(* CoDeSys 2.3.9.19 project: md_roman.pro *)
(* Libraries: D:\_wago\library\PowerMeasurement_01.lib 28.1.08 13:32:32, SysLibTime.lib 5.10.04 10:39:34, D:\_wago\library\Dali_01eng.lib 6.2.07 12:38:12, Building_common.lib 15.5.09 13:11:15, Util.lib 1.6.07 09:40:58, Standard.lib 22.11.04 11:21:12, SYSLIBCALLBACK.LIB 20.4.05 11:04:48 *)

(* PLC configuration (modules and I/O channels)
TL01 AT %IX17.0 [BOOLOnX_I] Vypinac_sklad_sklad
TL02 AT %IX17.1 [BOOLOnX_I] Vypinac_sklad_prodejna
TL03 AT %IX17.2 [BOOLOnX_I] Vypinac_sklad_z_venku
TL04 AT %IX17.3 [BOOLOnX_I] Vypinac_sklad_vrata_predni
TL05 AT %IX17.4 [BOOLOnX_I] Vypinac_sklad_vrata_zadni
TL06 AT %IX17.5 [BOOLOnX_I] Vypinac_prodejna_kolotoc_sude
TL07 AT %IX17.6 [BOOLOnX_I] Vypinac_prodejna_kolotoc_liche
TL08 AT %IX17.7 [BOOLOnX_I] Vypinac_prodejna_vypinac
TL09 AT %IX17.8 [BOOLOnX_I] Prodejna_Dali
TL10 AT %IX17.9 [BOOLOnX_I] Prodejna_faugule_OUT13
TL11 AT %IX17.10 [BOOLOnX_I] Ch_3 Digital input
TL12 AT %IX17.11 [BOOLOnX_I] Ch_4 Digital input
TL13 AT %IX17.12 [BOOLOnX_I] Ch_5 Digital input
AT %IX17.13 [BOOLOnX_I] Ch_6 Digital input
AT %IX17.14 [BOOLOnX_I] Ch_7 Digital input
AT %IX17.15 [BOOLOnX_I] Ch_8 Digital input
0750-0430 8 DI 24 V DC 3.0ms [Type_1_8_Channels] node 2, in %IB2 out %QB2 {INTTypePAAssignment = PLC; INTTypeModule = plugged}
  AT %IX18.0 [BOOLOnX_I] Ch_1 Digital input
  AT %IX18.1 [BOOLOnX_I] Ch_2 Digital input
  AT %IX18.2 [BOOLOnX_I] Ch_3 Digital input
  AT %IX18.3 [BOOLOnX_I] Ch_4 Digital input
  AT %IX18.4 [BOOLOnX_I] Ch_5 Digital input
  AT %IX18.5 [BOOLOnX_I] Ch_6 Digital input
  AT %IX18.6 [BOOLOnX_I] Ch_7 Digital input
  AT %IX18.7 [BOOLOnX_I] Ch_8 Digital input
0750-0530 8 DO 24 V DC 0.5A [Type_10_8_Channels] node 3, in %IB3 out %QB3 {INTTypePAAssignment = PLC; INTTypeModule = plugged}
  KA01 AT %QX9.0 [BOOLOnX_Q] Nevim
  KA02 AT %QX9.1 [BOOLOnX_Q] kolotoc2
  KA03 AT %QX9.2 [BOOLOnX_Q] kolotoc3
  KA04 AT %QX9.3 [BOOLOnX_Q] kolotoc4
  KA05 AT %QX9.4 [BOOLOnX_Q] kolotoc5
  KA06 AT %QX9.5 [BOOLOnX_Q] kolotoc6
  KA07 AT %QX9.6 [BOOLOnX_Q] kolotoc7
  KA08 AT %QX9.7 [BOOLOnX_Q] kolotoc8
0750-0530 8 DO 24 V DC 0.5A [Type_10_8_Channels] node 4, in %IB4 out %QB4 {INTTypePAAssignment = PLC; INTTypeModule = plugged}
  KA09 AT %QX9.8 [BOOLOnX_Q] kolotoc9
  KA10 AT %QX9.9 [BOOLOnX_Q] kolotoc10
  KA11 AT %QX9.10 [BOOLOnX_Q] kolotoc11
  KA12 AT %QX9.11 [BOOLOnX_Q] kolotoc12
  KA13 AT %QX9.12 [BOOLOnX_Q] svetlo_vchod_do_prodejny
  KA14 AT %QX9.13 [BOOLOnX_Q] reklama
  KA15 AT %QX9.14 [BOOLOnX_Q] svetlo_vrata_predni
  KA16 AT %QX9.15 [BOOLOnX_Q] svetlo_vrata_zadni
0750-0530 8 DO 24 V DC 0.5A [Type_10_8_Channels] node 5, in %IB5 out %QB5 {INTTypePAAssignment = PLC; INTTypeModule = plugged}
  KA17 AT %QX10.0 [BOOLOnX_Q] Ch_1 Digital output
  AT %QX10.1 [BOOLOnX_Q] Ch_2 Digital output
  AT %QX10.2 [BOOLOnX_Q] Ch_3 Digital output
  KA20 AT %QX10.3 [BOOLOnX_Q] Ch_4 Digital output
  AT %QX10.4 [BOOLOnX_Q] Ch_5 Digital output
  AT %QX10.5 [BOOLOnX_Q] Ch_6 Digital output
  AT %QX10.6 [BOOLOnX_Q] Ch_7 Digital output
  AT %QX10.7 [BOOLOnX_Q] Ch_8 Digital output
0750-0530 8 DO 24 V DC 0.5A [Type_10_8_Channels] node 6, in %IB6 out %QB6 {INTTypePAAssignment = PLC; INTTypeModule = plugged}
  AT %QX10.8 [BOOLOnX_Q] Ch_1 Digital output
  AT %QX10.9 [BOOLOnX_Q] Ch_2 Digital output
  AT %QX10.10 [BOOLOnX_Q] Ch_3 Digital output
  AT %QX10.11 [BOOLOnX_Q] Ch_4 Digital output
  AT %QX10.12 [BOOLOnX_Q] Ch_5 Digital output
  AT %QX10.13 [BOOLOnX_Q] Ch_6 Digital output
  AT %QX10.14 [BOOLOnX_Q] Ch_7 Digital output
  AT %QX10.15 [BOOLOnX_Q] Ch_8 Digital output
Analog_1 AT %IW0 [WORDOnW_I] Ch_1 Input word
AT %IW1 [WORDOnW_I] Ch_2 Input word
AT %IW2 [WORDOnW_I] Ch_3 Input word
AT %IW3 [WORDOnW_I] Ch_4 Input word
Teplota_1 AT %IW4 [INTOnW_I] Ch_1 signed Input value
Teplota_2 AT %IW5 [INTOnW_I] Ch_2 signed Input value
Teplota_3 AT %IW6 [INTOnW_I] Ch_3 signed Input value
Teplota_4 AT %IW7 [INTOnW_I] Ch_4 signed Input value
0750-0641 DALI/DSI-Master [Type_36_1_Channels] node 9, in %IB9 out %QB9 {INTTypePAAssignment = PLC; INTTypeModule = plugged}
  AT %IX8.0 [BOOLOnX_I] Transmit accepted
  AT %IX8.1 [BOOLOnX_I] Receive request
  AT %IX8.2 [BOOLOnX_I] Init accepted
  AT %IX8.3 [BOOLOnX_I] Actor Error
  AT %IX8.4 [BOOLOnX_I] Frame Error
  AT %IX8.5 [BOOLOnX_I] Bus Error
  AT %IX8.6 [BOOLOnX_I] General Module Error
  AT %IB17 [BYTEOnB_I] DALI Response
  AT %IB18 [BYTEOnB_I] DALI Address
  AT %IB19 [BYTEOnB_I] Message 3
  AT %IB20 [BYTEOnB_I] Message 2
  AT %IB21 [BYTEOnB_I] Message 1
  AT %QX0.0 [BOOLOnX_Q] Transmit request
  AT %QX0.1 [BOOLOnX_Q] Receive accepted
  AT %QX0.2 [BOOLOnX_Q] Init request
  AT %QB1 [BYTEOnB_Q] DALI Command, DSI dimming value
  AT %QB2 [BYTEOnB_Q] DALI Address
  AT %QB3 [BYTEOnB_Q] Parameter 2
  AT %QB4 [BYTEOnB_Q] Parameter 1
  AT %QB5 [BYTEOnB_Q] Command extension
fazeVstup AT %IB22 [BYTEOnB_I] First Byte of 12
fazeVystup AT %QB6 [BYTEOnB_Q] First Byte of 12
Fieldbus variables [FB_VARS] node 1, in %IB0 out %QB0
*)

(* Task configuration *)
TASK hlavni (PRIORITY := 1, INTERVAL := T#20ms);
	PLC_PRG();
END_TASK

(* Global variable list: Global_Variables *)
VAR_GLOBAL
	start_bit: BOOL;
	Inicialiazace_DALI: BOOL;
	Inicializuj: BOOL;
	TL08s: BOOL;
	TL07s: BOOL;
	TL10s: BOOL;
	TL06s: BOOL;
	TL05s: BOOL;
	TL01s: BOOL;
	TL09s: BOOL;
END_VAR

(* POU PLC_PRG, FBD *)
PROGRAM PLC_PRG
VAR
	cas_datum: CurTimeEx;
	System_cas: SysTime64;
	System_datum: SystemTimeDate;
	kolotoc1: kolotoc;
	kolotoc2: kolotoc;
	BLINK_nouzaky: BLINK;
	LibovolnyVystup: BOOL;
END_VAR
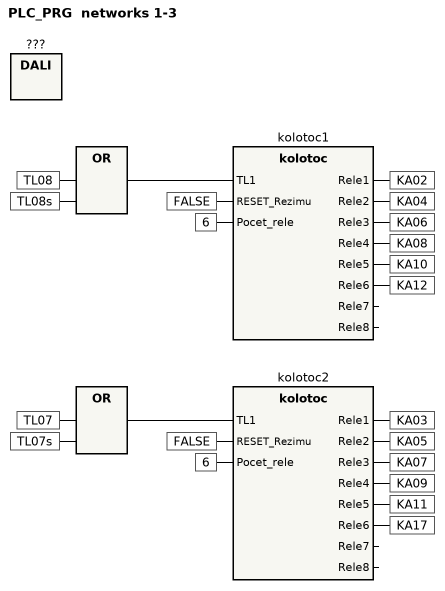
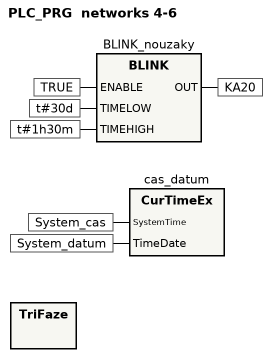
_FBD_ (* Function Block Diagram *)
NETWORK 1
	???:DALI()
NETWORK 2
	kolotoc1:kolotoc(TL1: OR(TL08, TL08s), RESET_Rezimu: FALSE, Pocet_rele: 6, Rele2 => KA04, Rele3 => KA06, Rele4 => KA08, Rele5 => KA10, Rele6 => KA12) => KA02
NETWORK 3
	kolotoc2:kolotoc(TL1: OR(TL07, TL07s), RESET_Rezimu: FALSE, Pocet_rele: 6, Rele2 => KA05, Rele3 => KA07, Rele4 => KA09, Rele5 => KA11, Rele6 => KA17) => KA03
NETWORK 4
	BLINK_nouzaky:BLINK(ENABLE: TRUE, TIMELOW: t#30d, TIMEHIGH: t#1h30m) => KA20
NETWORK 5
	cas_datum:CurTimeEx(SystemTime: System_cas, TimeDate: System_datum)
NETWORK 6
	TriFaze()
_END_FBD_
(* the same logic as Structured Text *)
(* Network 1: see the listing above *)
(* Network 2 *)
kolotoc1(TL1 := TL08 OR TL08s, RESET_Rezimu := FALSE, Pocet_rele := 6);
KA04 := kolotoc1.Rele2;
KA06 := kolotoc1.Rele3;
KA08 := kolotoc1.Rele4;
KA10 := kolotoc1.Rele5;
KA12 := kolotoc1.Rele6;
KA02 := kolotoc1.Rele1;
(* Network 3 *)
kolotoc2(TL1 := TL07 OR TL07s, RESET_Rezimu := FALSE, Pocet_rele := 6);
KA05 := kolotoc2.Rele2;
KA07 := kolotoc2.Rele3;
KA09 := kolotoc2.Rele4;
KA11 := kolotoc2.Rele5;
KA17 := kolotoc2.Rele6;
KA03 := kolotoc2.Rele1;
(* Network 4 *)
BLINK_nouzaky(ENABLE := TRUE, TIMELOW := t#30d, TIMEHIGH := t#1h30m);
KA20 := BLINK_nouzaky.OUT;
(* Network 5 *)
cas_datum(SystemTime := System_cas, TimeDate := System_datum);
(* Network 6 *)
TriFaze();
END_PROGRAM

(* POU dali/kolotoc, FBD *)
FUNCTION_BLOCK kolotoc
VAR
	Data_platna: BOOL;
	Data_platna_reset: BOOL;
	T_Data_platna: TON;
	T_Data_platna_reset: TON;
	Stisk_kratky: BOOL := FALSE;
	Stisk_dlouhy: BOOL := FALSE;
	T_stisk_TLx: TON;
	F_trig_hr1: F_TRIG;
	R_trig_hr2: R_TRIG;
	TL1_Citac: CTU;
	SR_stisk_TLx: SR;
	ZAP_VYP: BOOL;




	TP_byl_kratky: TP;
	Q_byl_kratky: BOOL;
	blok_kratky: BOOL;
	TL1_hr1: BOOL;
	SET_stisk_TL1: BOOL;
	Q_stisk_TL1: BOOL;
	TL1_INT: INT;
END_VAR

VAR_OUTPUT
	Rele1: BOOL;
	Rele2: BOOL;
	Rele3: BOOL;
	Rele4: BOOL;
	Rele5: BOOL;
	Rele6: BOOL;
	Rele7: BOOL;
	Rele8: BOOL;
END_VAR
VAR_INPUT
	TL1: BOOL;
	RESET_Rezimu: BOOL;
	Pocet_rele: INT;
END_VAR
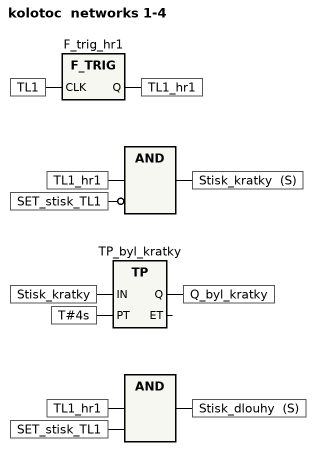
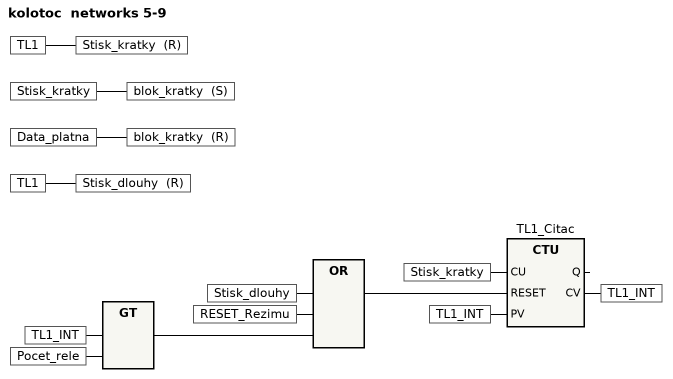
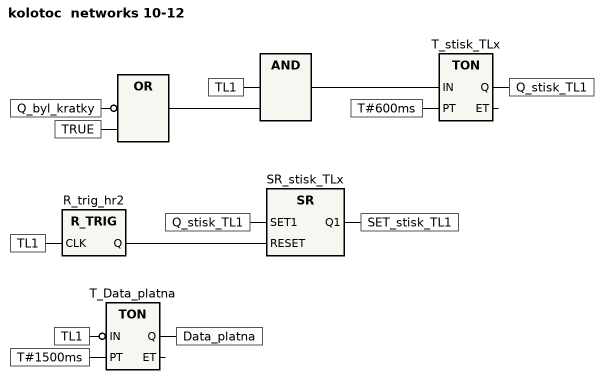
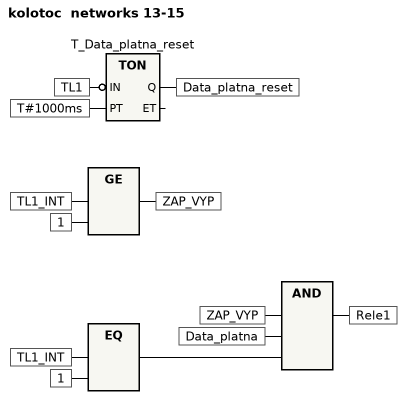
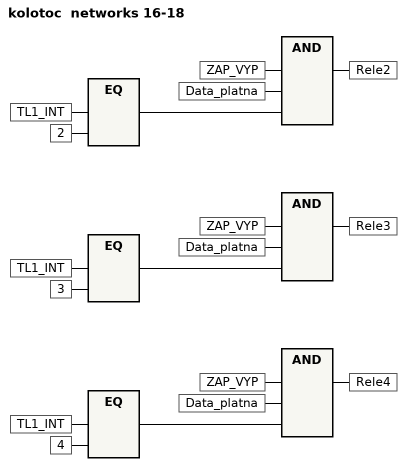
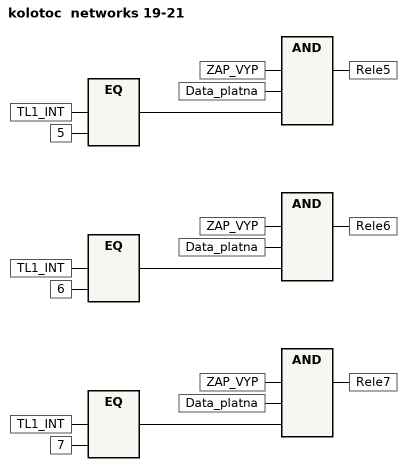
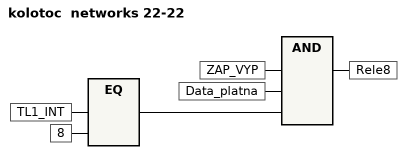
_FBD_ (* Function Block Diagram *)
NETWORK 1
	F_trig_hr1:F_TRIG(CLK: TL1) => TL1_hr1
NETWORK 2
	AND(TL1_hr1, NOT SET_stisk_TL1) => S Stisk_kratky
NETWORK 3
	TP_byl_kratky:TP(IN: Stisk_kratky, PT: T#4s) => Q_byl_kratky
NETWORK 4
	AND(TL1_hr1, SET_stisk_TL1) => S Stisk_dlouhy
NETWORK 5
	TL1 => R Stisk_kratky
NETWORK 6
	Stisk_kratky => S blok_kratky
NETWORK 7
	Data_platna => R blok_kratky
NETWORK 8
	TL1 => R Stisk_dlouhy
NETWORK 9
	TL1_Citac:CTU(CU: Stisk_kratky, RESET: OR(Stisk_dlouhy, RESET_Rezimu, GT(TL1_INT, Pocet_rele)), PV: TL1_INT, CV => TL1_INT)
NETWORK 10 (* delka stisku TLx *)
	T_stisk_TLx:TON(IN: AND(TL1, OR(NOT Q_byl_kratky, TRUE)), PT: T#600ms) => Q_stisk_TL1
NETWORK 11
	SR_stisk_TLx:SR(SET1: Q_stisk_TL1, RESET: R_trig_hr2:R_TRIG(CLK: TL1)) => SET_stisk_TL1
NETWORK 12 (* Data platna *)
	T_Data_platna:TON(IN: NOT TL1, PT: T#1500ms) => Data_platna
NETWORK 13 (* Data platna *)
	T_Data_platna_reset:TON(IN: NOT TL1, PT: T#1000ms) => Data_platna_reset
NETWORK 14
	GE(TL1_INT, 1) => ZAP_VYP
NETWORK 15
	AND(ZAP_VYP, Data_platna, EQ(TL1_INT, 1)) => Rele1
NETWORK 16
	AND(ZAP_VYP, Data_platna, EQ(TL1_INT, 2)) => Rele2
NETWORK 17
	AND(ZAP_VYP, Data_platna, EQ(TL1_INT, 3)) => Rele3
NETWORK 18
	AND(ZAP_VYP, Data_platna, EQ(TL1_INT, 4)) => Rele4
NETWORK 19
	AND(ZAP_VYP, Data_platna, EQ(TL1_INT, 5)) => Rele5
NETWORK 20
	AND(ZAP_VYP, Data_platna, EQ(TL1_INT, 6)) => Rele6
NETWORK 21
	AND(ZAP_VYP, Data_platna, EQ(TL1_INT, 7)) => Rele7
NETWORK 22
	AND(ZAP_VYP, Data_platna, EQ(TL1_INT, 8)) => Rele8
_END_FBD_
(* the same logic as Structured Text *)
(* Network 1 *)
F_trig_hr1(CLK := TL1);
TL1_hr1 := F_trig_hr1.Q;
(* Network 2 *)
IF TL1_hr1 AND NOT SET_stisk_TL1 THEN Stisk_kratky := TRUE; END_IF;
(* Network 3 *)
TP_byl_kratky(IN := Stisk_kratky, PT := T#4s);
Q_byl_kratky := TP_byl_kratky.Q;
(* Network 4 *)
IF TL1_hr1 AND SET_stisk_TL1 THEN Stisk_dlouhy := TRUE; END_IF;
(* Network 5 *)
IF TL1 THEN Stisk_kratky := FALSE; END_IF;
(* Network 6 *)
IF Stisk_kratky THEN blok_kratky := TRUE; END_IF;
(* Network 7 *)
IF Data_platna THEN blok_kratky := FALSE; END_IF;
(* Network 8 *)
IF TL1 THEN Stisk_dlouhy := FALSE; END_IF;
(* Network 9 *)
TL1_Citac(CU := Stisk_kratky, RESET := Stisk_dlouhy OR RESET_Rezimu OR (TL1_INT > Pocet_rele), PV := TL1_INT);
TL1_INT := TL1_Citac.CV;
(* Network 10: see the listing above *)
(* Network 11 *)
R_trig_hr2(CLK := TL1);
SR_stisk_TLx(SET1 := Q_stisk_TL1, RESET := R_trig_hr2.Q);
SET_stisk_TL1 := SR_stisk_TLx.Q1;
(* Network 12 *)
T_Data_platna(IN := NOT TL1, PT := T#1500ms);
Data_platna := T_Data_platna.Q;
(* Network 13 *)
T_Data_platna_reset(IN := NOT TL1, PT := T#1000ms);
Data_platna_reset := T_Data_platna_reset.Q;
(* Network 14 *)
ZAP_VYP := TL1_INT >= 1;
(* Network 15 *)
Rele1 := ZAP_VYP AND Data_platna AND (TL1_INT = 1);
(* Network 16 *)
Rele2 := ZAP_VYP AND Data_platna AND (TL1_INT = 2);
(* Network 17 *)
Rele3 := ZAP_VYP AND Data_platna AND (TL1_INT = 3);
(* Network 18 *)
Rele4 := ZAP_VYP AND Data_platna AND (TL1_INT = 4);
(* Network 19 *)
Rele5 := ZAP_VYP AND Data_platna AND (TL1_INT = 5);
(* Network 20 *)
Rele6 := ZAP_VYP AND Data_platna AND (TL1_INT = 6);
(* Network 21 *)
Rele7 := ZAP_VYP AND Data_platna AND (TL1_INT = 7);
(* Network 22 *)
Rele8 := ZAP_VYP AND Data_platna AND (TL1_INT = 8);
END_FUNCTION_BLOCK

(* POU dali/DALI, FBD *)
PROGRAM DALI
VAR
	trojklik_sklad: Trojklik;
	D_M: FbDALI_Joblist;
	In_data AT %IB16: ARRAY [0..5] OF BYTE;
	Out_data AT %QB0: ARRAY [0..5] OF BYTE;
	Jobs: typDaliJoblisten;
	short_group: BOOL := FALSE;
	hodnota_po_zapnuti: BYTE := 50;
	hodnota_po_zapnuti_prodejna: BYTE := 100;
	povolit_vypnuti_pri_minimum: BOOL := FALSE;
	rychlost_zneny: BYTE := 7;
	co_je_kratky_a_dlouhy_stisk: BYTE := 6;
      OP_reset1: BOOL;
	OP_reset2: BOOL;
	OP_reset3: BOOL;
	OP_reset_OUT15: BOOL;
	OP_reset_OUT16: BOOL;

	Svetlo_adr1: FbDALI_Latching_Relay;
	Svetlo_adr2: FbDALI_Latching_Relay;
	Svetlo_adr3: FbDALI_Latching_Relay;
	Svetlo_adr4: FbDALI_Dimm_Single_Switch;

	stav_adr1: BYTE;
	stav_adr2: BYTE;
	stav_adr3: BYTE;
	stav_adr4: BYTE;


	trojklik_prodejna: Trojklik;
	OP_reset4: BOOL;
	Trojklik_Fagule_OUT13: Trojklik;
	OP_reset5: BOOL;
	TP_ALL: TP;
	Q_All: BOOL;
	Dali_Status_03: FbDALI_Status_DimmValue;
	dali_status_Ready03: BOOL;
	dali_status_Feedback03: BYTE;
	dali_status_Status03: BOOL;
	dali_DimmValue_Ready03: BYTE;
	Reset_ini: TON;
	Dali_Status_09: FbDALI_Status_DimmValue;
	dali_status_Ready09: BOOL;
	dali_status_Feedback09: BYTE;
	dali_status_Status09: BOOL;
	dali_DimmValue_Ready09: BYTE;
	Dali_Status_19: FbDALI_Status_DimmValue;
	dali_status_Ready19: BOOL;
	dali_status_Feedback19: BYTE;
	dali_status_Status19: BOOL;
	dali_DimmValue_Ready19: BYTE;
	TON_ALL: TON;
	pom1: BOOL;
	go: BOOL;


	Fb_ShortLong1: Fb_ShortLong;
	CTU1: CTU;
	R_TRIG1: R_TRIG;
	TP1: TP;
	F_TRIG1: F_TRIG;
	STAV: WORD;
	CasNaKlik: TIME := t#1s500ms;
	F_TRIG2: F_TRIG;
	R_TRIG2: R_TRIG;
	Zhasni1: Zhasni;
	F_TRIG3: F_TRIG;
	Fb_LatchingRelay1: Fb_LatchingRelay;
	KratkyKlik: BOOL;
	Fb_ShortLong2: Fb_ShortLong;
	Fb_LatchingRelay2: Fb_LatchingRelay;
	Fb_ShortLong3: Fb_ShortLong;
	KratkyKlikA: BOOL;
	KratkyKlikB: BOOL;
	KratkyKlikC: BOOL;
	Svetlo_adr_255: FbDALI_Latching_Relay;
	stav_adr255: BYTE;
	TON_Cental_Off: TON;
	R_TRIG6: R_TRIG;
	ka15cas: TON;
	ka15pink: TP;
	TL06p: BOOL;
	ka16cas: TON;
	ka16pink: TP;
	TL05p: BOOL;
	ka13cas: TON;
	ka13pink: TP;
 	TL10p: BOOL;
	casvensvetel: TIME:= t#10m;
END_VAR
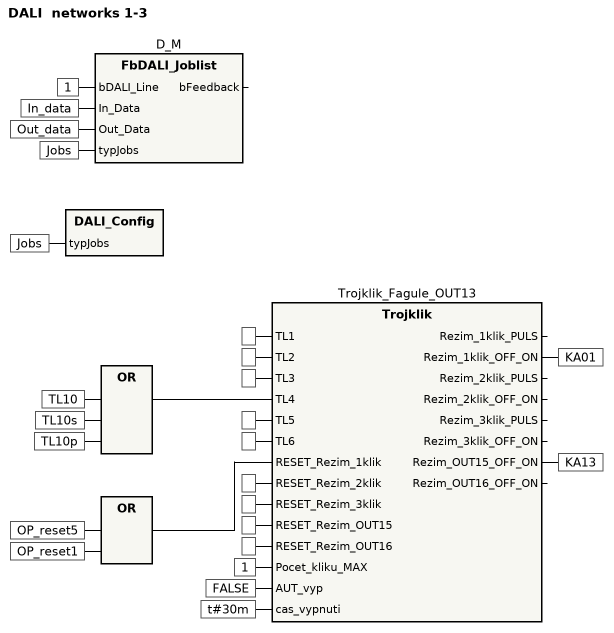
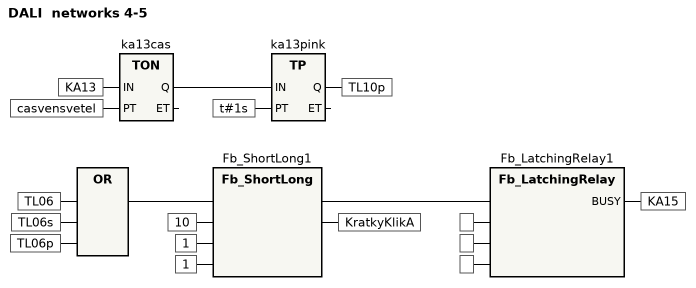
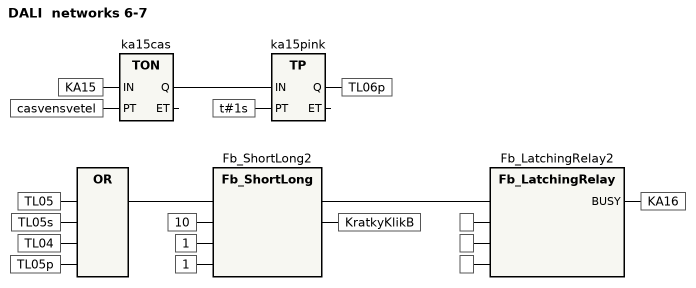
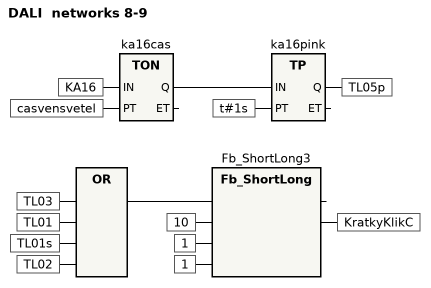
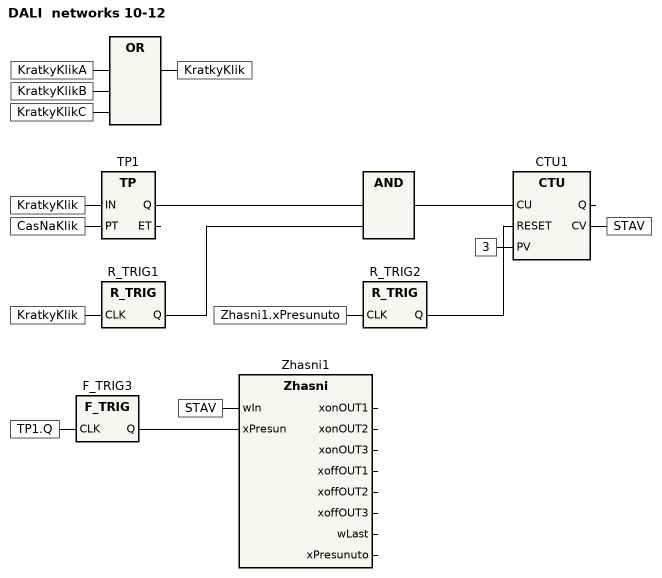
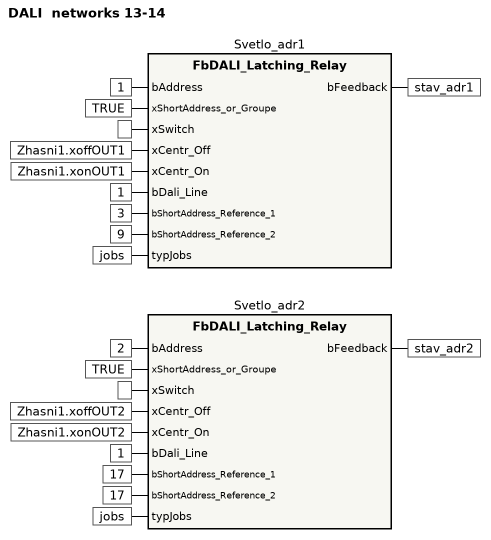
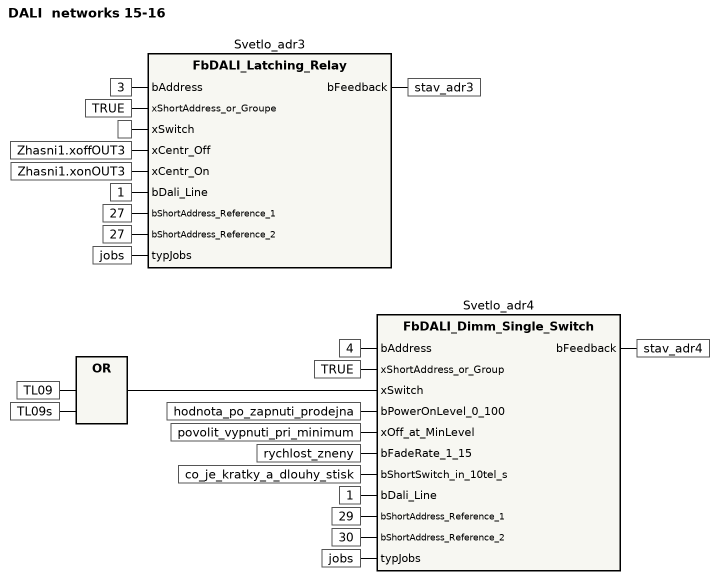
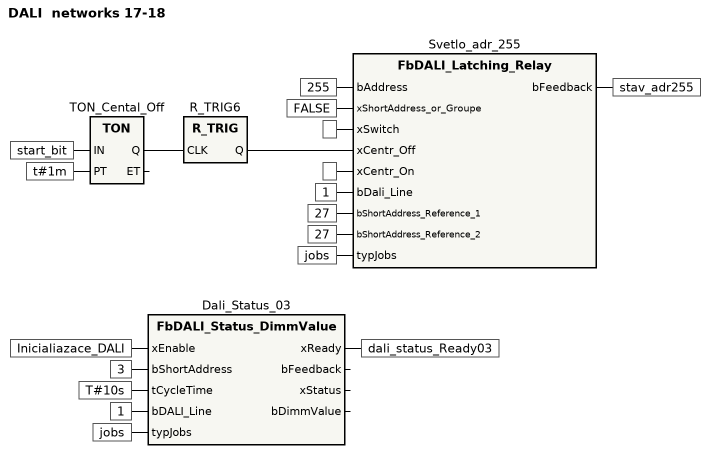
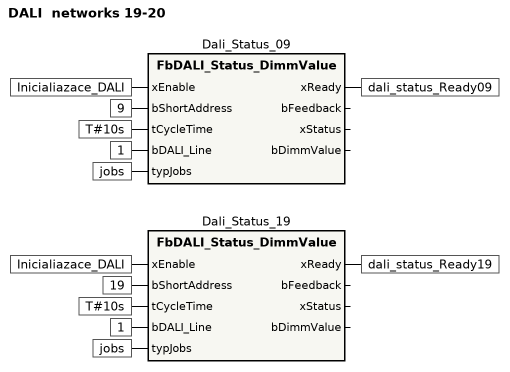
_FBD_ (* Function Block Diagram *)
NETWORK 1
	D_M:FbDALI_Joblist(bDALI_Line: 1, In_Data: In_data, Out_Data: Out_data, typJobs: Jobs)
NETWORK 2
	DALI_Config(typJobs: Jobs)
NETWORK 3
	Trojklik_Fagule_OUT13:Trojklik(TL1: , TL2: , TL3: , TL4: OR(TL10, TL10s, TL10p), TL5: , TL6: , RESET_Rezim_1klik: OR(OP_reset5, OP_reset1), RESET_Rezim_2klik: , RESET_Rezim_3klik: , RESET_Rezim_OUT15: , RESET_Rezim_OUT16: , Pocet_kliku_MAX: 1, AUT_vyp: FALSE, cas_vypnuti: t#30m, Rezim_1klik_OFF_ON => KA01, Rezim_OUT15_OFF_ON => KA13)
NETWORK 4
	ka13pink:TP(IN: ka13cas:TON(IN: KA13, PT: casvensvetel), PT: t#1s) => TL10p
NETWORK 5
	Fb_LatchingRelay1:Fb_LatchingRelay(Fb_ShortLong1:Fb_ShortLong(OR(TL06, TL06s, TL06p), 10, 1, 1, out 2 => KratkyKlikA), , , ) => KA15
NETWORK 6
	ka15pink:TP(IN: ka15cas:TON(IN: KA15, PT: casvensvetel), PT: t#1s) => TL06p
NETWORK 7
	Fb_LatchingRelay2:Fb_LatchingRelay(Fb_ShortLong2:Fb_ShortLong(OR(TL05, TL05s, TL04, TL05p), 10, 1, 1, out 2 => KratkyKlikB), , , ) => KA16
NETWORK 8
	ka16pink:TP(IN: ka16cas:TON(IN: KA16, PT: casvensvetel), PT: t#1s) => TL05p
NETWORK 9
	Fb_ShortLong3:Fb_ShortLong(OR(TL03, TL01, TL01s, TL02), 10, 1, 1, out 2 => KratkyKlikC)
NETWORK 10
	OR(KratkyKlikA, KratkyKlikB, KratkyKlikC) => KratkyKlik
NETWORK 11
	CTU1:CTU(CU: AND(TP1:TP(IN: KratkyKlik, PT: CasNaKlik), R_TRIG1:R_TRIG(CLK: KratkyKlik)), RESET: R_TRIG2:R_TRIG(CLK: Zhasni1.xPresunuto), PV: 3, CV => STAV)
NETWORK 12
	Zhasni1:Zhasni(wIn: STAV, xPresun: F_TRIG3:F_TRIG(CLK: TP1.Q))
NETWORK 13
	Svetlo_adr1:FbDALI_Latching_Relay(bAddress: 1, xShortAddress_or_Groupe: TRUE, xSwitch: , xCentr_Off: Zhasni1.xoffOUT1, xCentr_On: Zhasni1.xonOUT1, bDali_Line: 1, bShortAddress_Reference_1: 3, bShortAddress_Reference_2: 9, typJobs: jobs) => stav_adr1
NETWORK 14
	Svetlo_adr2:FbDALI_Latching_Relay(bAddress: 2, xShortAddress_or_Groupe: TRUE, xSwitch: , xCentr_Off: Zhasni1.xoffOUT2, xCentr_On: Zhasni1.xonOUT2, bDali_Line: 1, bShortAddress_Reference_1: 17, bShortAddress_Reference_2: 17, typJobs: jobs) => stav_adr2
NETWORK 15
	Svetlo_adr3:FbDALI_Latching_Relay(bAddress: 3, xShortAddress_or_Groupe: TRUE, xSwitch: , xCentr_Off: Zhasni1.xoffOUT3, xCentr_On: Zhasni1.xonOUT3, bDali_Line: 1, bShortAddress_Reference_1: 27, bShortAddress_Reference_2: 27, typJobs: jobs) => stav_adr3
NETWORK 16
	Svetlo_adr4:FbDALI_Dimm_Single_Switch(bAddress: 4, xShortAddress_or_Group: TRUE, xSwitch: OR(TL09, TL09s), bPowerOnLevel_0_100: hodnota_po_zapnuti_prodejna, xOff_at_MinLevel: povolit_vypnuti_pri_minimum, bFadeRate_1_15: rychlost_zneny, bShortSwitch_in_10tel_s: co_je_kratky_a_dlouhy_stisk, bDali_Line: 1, bShortAddress_Reference_1: 29, bShortAddress_Reference_2: 30, typJobs: jobs) => stav_adr4
NETWORK 17 (* Po 1min po restartu dojde k vypnuti vsech svitidel *)
	Svetlo_adr_255:FbDALI_Latching_Relay(bAddress: 255, xShortAddress_or_Groupe: FALSE, xSwitch: , xCentr_Off: R_TRIG6:R_TRIG(CLK: TON_Cental_Off:TON(IN: start_bit, PT: t#1m)), xCentr_On: , bDali_Line: 1, bShortAddress_Reference_1: 27, bShortAddress_Reference_2: 27, typJobs: jobs) => stav_adr255
NETWORK 18
	Dali_Status_03:FbDALI_Status_DimmValue(xEnable: Inicialiazace_DALI, bShortAddress: 3, tCycleTime: T#10s, bDALI_Line: 1, typJobs: jobs) => dali_status_Ready03
NETWORK 19
	Dali_Status_09:FbDALI_Status_DimmValue(xEnable: Inicialiazace_DALI, bShortAddress: 9, tCycleTime: T#10s, bDALI_Line: 1, typJobs: jobs) => dali_status_Ready09
NETWORK 20
	Dali_Status_19:FbDALI_Status_DimmValue(xEnable: Inicialiazace_DALI, bShortAddress: 19, tCycleTime: T#10s, bDALI_Line: 1, typJobs: jobs) => dali_status_Ready19
_END_FBD_
(* the same logic as Structured Text *)
(* Network 1 *)
D_M(bDALI_Line := 1, In_Data := In_data, Out_Data := Out_data, typJobs := Jobs);
(* Network 2 *)
DALI_Config(typJobs := Jobs);
(* Network 3: see the listing above *)
(* Network 4 *)
ka13cas(IN := KA13, PT := casvensvetel);
ka13pink(IN := ka13cas.Q, PT := t#1s);
TL10p := ka13pink.Q;
(* Network 5: see the listing above *)
(* Network 6 *)
ka15cas(IN := KA15, PT := casvensvetel);
ka15pink(IN := ka15cas.Q, PT := t#1s);
TL06p := ka15pink.Q;
(* Network 7: see the listing above *)
(* Network 8 *)
ka16cas(IN := KA16, PT := casvensvetel);
ka16pink(IN := ka16cas.Q, PT := t#1s);
TL05p := ka16pink.Q;
(* Network 9: see the listing above *)
(* Network 10 *)
KratkyKlik := KratkyKlikA OR KratkyKlikB OR KratkyKlikC;
(* Network 11 *)
TP1(IN := KratkyKlik, PT := CasNaKlik);
R_TRIG1(CLK := KratkyKlik);
R_TRIG2(CLK := Zhasni1.xPresunuto);
CTU1(CU := TP1.Q AND R_TRIG1.Q, RESET := R_TRIG2.Q, PV := 3);
STAV := CTU1.CV;
(* Network 12 *)
F_TRIG3(CLK := TP1.Q);
Zhasni1(wIn := STAV, xPresun := F_TRIG3.Q);
(* Network 13: see the listing above *)
(* Network 14: see the listing above *)
(* Network 15: see the listing above *)
(* Network 16 *)
Svetlo_adr4(bAddress := 4, xShortAddress_or_Group := TRUE, xSwitch := TL09 OR TL09s, bPowerOnLevel_0_100 := hodnota_po_zapnuti_prodejna, xOff_at_MinLevel := povolit_vypnuti_pri_minimum, bFadeRate_1_15 := rychlost_zneny, bShortSwitch_in_10tel_s := co_je_kratky_a_dlouhy_stisk, bDali_Line := 1, bShortAddress_Reference_1 := 29, bShortAddress_Reference_2 := 30, typJobs := jobs);
stav_adr4 := Svetlo_adr4.bFeedback;
(* Network 17: see the listing above *)
(* Network 18 *)
Dali_Status_03(xEnable := Inicialiazace_DALI, bShortAddress := 3, tCycleTime := T#10s, bDALI_Line := 1, typJobs := jobs);
dali_status_Ready03 := Dali_Status_03.xReady;
(* Network 19 *)
Dali_Status_09(xEnable := Inicialiazace_DALI, bShortAddress := 9, tCycleTime := T#10s, bDALI_Line := 1, typJobs := jobs);
dali_status_Ready09 := Dali_Status_09.xReady;
(* Network 20 *)
Dali_Status_19(xEnable := Inicialiazace_DALI, bShortAddress := 19, tCycleTime := T#10s, bDALI_Line := 1, typJobs := jobs);
dali_status_Ready19 := Dali_Status_19.xReady;
END_PROGRAM

(* POU dali/Trojklik, FBD *)
FUNCTION_BLOCK Trojklik
VAR
	TLx_sklad: BOOL;
	Data_platna: BOOL;
	Data_platna_reset: BOOL;
	T_Data_platna: TON;
	T_Data_platna_reset: TON;
	Stisk_kratky: BOOL := FALSE;
	Stisk_dlouhy: BOOL := FALSE;
	Q_stisk_TLx: BOOL;
	T_stisk_TLx: TON;
	F_trig_hr1: F_TRIG;
	R_trig_hr2: R_TRIG;
	TLx_sklad_hr1: BOOL;
	TLx_INT: INT;
	TLx_Citac: CTU;
	SET_stisk_TLx: BOOL;
	SR_stisk_TLx: SR;

	ZAP_VYP_sklad: BOOL;
	mod_1klik: BOOL;
	mod_2klik: BOOL;
	blok: BOOL;
	blok_ZAP_VYP: BOOL;
	T_blok: TON;
	T_blok_ZAP_VYP: TON;
	TP_mode_1klik: TP;

	TP_mode_2klik: TP;

	TP_byl_kratky: TP;
	Q_byl_kratky: BOOL;
	blok_kratky: BOOL;
	mod_3klik: BOOL;
	TP_mode_3klik: TP;

	TP_reset1: TP;
	TP_reset2: TP;
	TP_reset3: TP;
	TLx_zvenku: BOOL;
	T_stisk_TLx_zvenku: TON;
	TLx_sklad_hr1_zvenku: BOOL;
	F_trig_hr1_zvenku: F_TRIG;
	Stisk_kratky_zvenku: BOOL;
	SET_stisk_TLx_zvenku: BOOL;
	Q_byl_kratky_zvenku: BOOL;
	TP_byl_kratky_zvenku: TP;
	Stisk_dlouhy_zvenku: BOOL;
	blok_kratky_zvenku: BOOL;
	TLx_INT_zvenku: INT;
	TLx_Citac_zvenku: CTU;
	Q_stisk_TLx_zvenku: BOOL;
	R_trig_hr2_zvenku: R_TRIG;
	SR_stisk_TLx_zvenku: SR;
	blok_OUT15: BOOL;
	TOF_OUT15_zp: TOF;
	R_trig_OUT15: R_TRIG;
	R_trig_OUT15b: R_TRIG;
	TON_blok_OUT15: TON;
	TON_AUT_stop_OUT15: TON;
	R_trig_OUT16: R_TRIG;
	TOF_OUT16_zp: TOF;
	blok_OUT16: BOOL;
	R_trig_OUT16b: R_TRIG;
	TON_AUT_stop_OUT16: TON;
	TON_blok_OUT16: TON;
	T_max: TON;
	Q_T_MAX: BOOL;
	TP_T_max: TP;
	Aktivni_TL1: BOOL;
	Aktivni_TL2: BOOL;
	Aktivni_TL3: BOOL;
	Aktivni_TL4: BOOL;
	Aktivni_TL5: BOOL;
	Aktivni_TL6: BOOL;
	T_vypnuti_ukonceno: TP;
	Q_vypnuti_ukonceno: BOOL;
	F_trig_1klik: F_TRIG;
	F_trig_2klik: F_TRIG;
	F_trig_3klik: F_TRIG;
	tp_1klik_vyp: TP;
	f_trig_1klik_vyp: F_TRIG;
	tp_2klik_vyp: TP;
	f_trig_2klik_vyp: F_TRIG;
	f_trig_3klik_vyp: F_TRIG;
	tp_3klik_vyp: TP;
END_VAR

VAR_OUTPUT
	Rezim_1klik_PULS: BOOL;
	Rezim_1klik_OFF_ON: BOOL;
	Rezim_2klik_PULS: BOOL;
	Rezim_2klik_OFF_ON: BOOL;
	Rezim_3klik_PULS: BOOL;
	Rezim_3klik_OFF_ON: BOOL;
	Rezim_OUT15_OFF_ON: BOOL;
	Rezim_OUT16_OFF_ON: BOOL;
END_VAR
VAR_INPUT
	TL1: BOOL;
	TL2: BOOL;
	TL3: BOOL;
	TL4: BOOL;
	TL5: BOOL;
	TL6: BOOL;
	RESET_Rezim_1klik: BOOL;
	RESET_Rezim_2klik: BOOL;
	RESET_Rezim_3klik: BOOL;
	RESET_Rezim_OUT15: BOOL;
	RESET_Rezim_OUT16: BOOL;
	Pocet_kliku_MAX: INT;
	AUT_vyp: BOOL;
	cas_vypnuti: TIME;
END_VAR
VAR (* helpers for the ST form of the networks *)
	_p1 : BOOL;
	_p2 : BOOL;
	_p3 : BOOL;
	_p4 : BOOL;
	_p5 : BOOL;
	_p6 : BOOL;
	_p7 : BOOL;
END_VAR
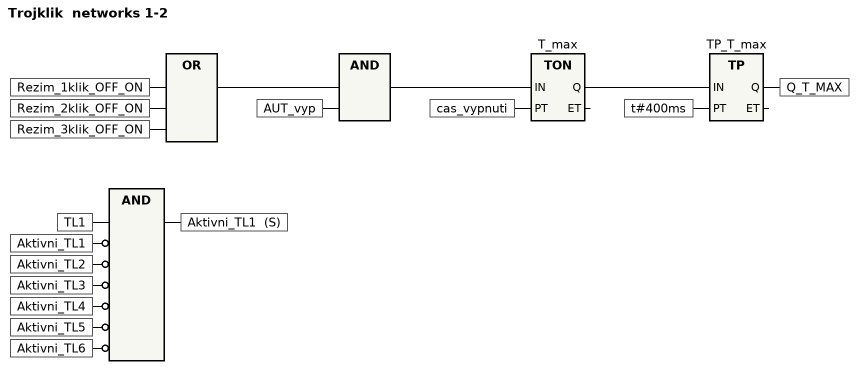
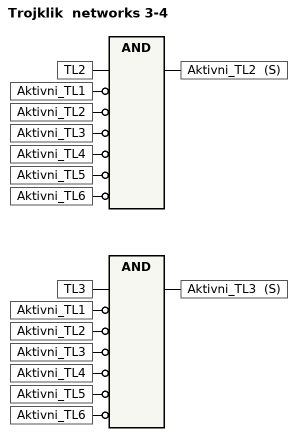
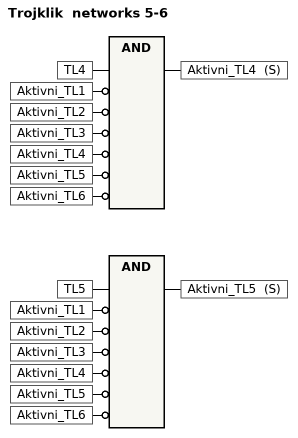
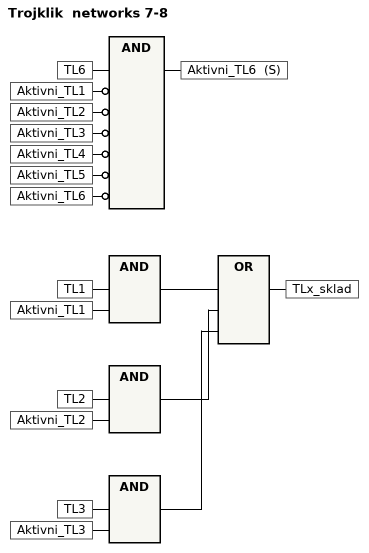
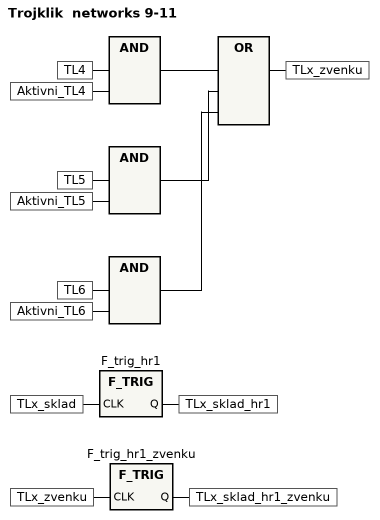
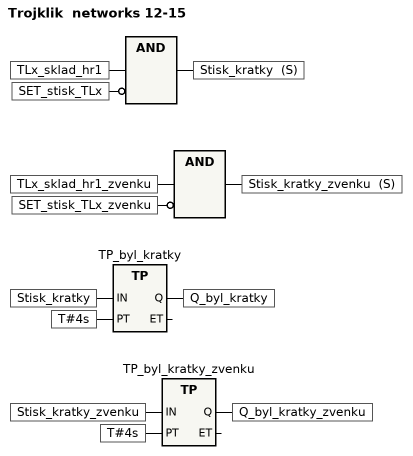
